ABB RobotStudio station: RobotStudio_PickAndGo.rspag

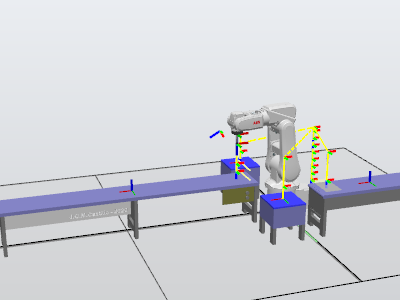
--- station ---
Station Project1 (saved by RobotStudio 24.4.11080.0)
Controller Controlador_1
  mechanical unit ROB_1: IRB120_3_58__01, 6 joints, base frame (0, 0, 0) mm
Layout (positions relative to the parent item):
  - IRB120_3_58__01 [mechanism, from %ABB.RobotStudio.Models.IRB120%\IRB120_3_58_G_01.rslib] at (0, 0, 0) mm; joint values [0.1232, 0.0796, -0.0396, 0, 1.5308, 0.1232] (rad or m)
  - CintaConveyor [protected smart component, left out]
  - CintaDescarga [protected smart component, left out]
  - Caja IZQ [protected smart component, left out]
  - Ventosa [protected smart component, left out]
  - Caja DER [protected smart component, left out]
Attachment: Ventosa is attached to IRB120_3_58__01 / Link6
Attachment: Workobject_Conveyor is attached to Belt
Attachment: Workobject_Mesa1 is attached to Tapa
Attachment: Workobject_CintaDescarga is attached to Cinta de transporte
Attachment: Workobject_Mesa2 is attached to Tapa
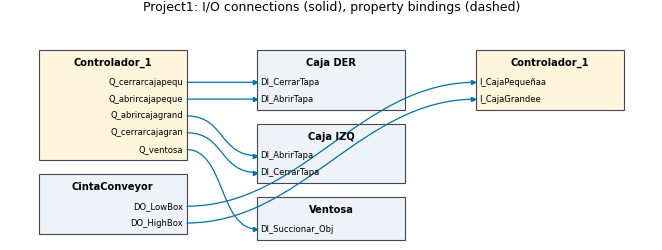
Station logic (signal -> signal, property => property):
  Controlador_1.Q_cerrarcajapequeña -> Caja DER.DI_CerrarTapa
  Controlador_1.Q_abrircajapequeña -> Caja DER.DI_AbrirTapa
  Controlador_1.Q_abrircajagrande -> Caja IZQ.DI_AbrirTapa
  Controlador_1.Q_cerrarcajagrande -> Caja IZQ.DI_CerrarTapa
  Controlador_1.Q_ventosa -> Ventosa.DI_Succionar_Objeto
  CintaConveyor.DO_LowBox -> Controlador_1.I_CajaPequeñaa
  CintaConveyor.DO_HighBox -> Controlador_1.I_CajaGrandee
Targets, tools, work objects and paths stored in the station and not in the controller backup, written as RAPID:
! task T_ROB1
MODULE Module1
  PROC setup()
    MoveJ Target_10,velocidad,z0,TCP_Ventosa\WObj:=wobj0;
  ENDPROC
ENDMODULE

! task T_ROB1
MODULE Rutinas_eventos
  PROC Paro_off()
    SetDO Q_Paro,0;
  ENDPROC
  PROC Paro_on()
    SetDO Q_Paro,1;
  ENDPROC
  PROC Power_Controladora()
    SetDO Q_Power_Controladora,1;
  ENDPROC
ENDMODULE


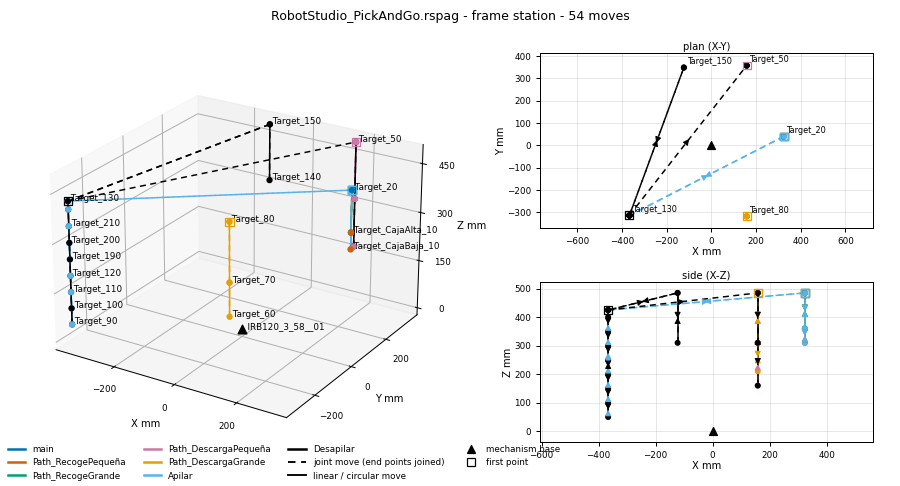
[picture p0: tool path of RobotStudio_PickAndGo.rspag in frame station, 54 of 54 moves have a stored position in this frame; points joined in program order, loops and branches not executed]
--- Controller Data/Controlador_1/RAPID/TASK1/PROGMOD/CalibData.mod ---
MODULE CalibData
    PERS tooldata TCP_Ventosa:=[TRUE,[[0,0,60],[1,0,0,0]],[0.1,[0,0,1],[1,0,0,0],0,0,0]];
    TASK PERS wobjdata Workobject_Conveyor:=[FALSE,TRUE,"",[[971.48,35.469,260],[1,0,0,0]],[[0,0,0],[1,0,0,0]]];
    TASK PERS wobjdata Workobject_Mesa1:=[FALSE,TRUE,"",[[158.333,357.694,230],[1,0,0,0]],[[0,0,0],[1,0,0,0]]];
    TASK PERS wobjdata Workobject_Mesa2:=[FALSE,TRUE,"",[[158.333,-317.306,230],[1,0,0,0]],[[0,0,0],[1,0,0,0]]];
    TASK PERS wobjdata Workobject_CintaDescarga:=[FALSE,TRUE,"",[[-411.761,348.55,260],[1,0,0,0]],[[0,0,0],[1,0,0,0]]];
    TASK PERS wobjdata Workobject_Apilar:=[FALSE,TRUE,"",[[-366.457,-313.205,0],[1,0,0,0]],[[0,0,0],[1,0,0,0]]];
ENDMODULE

--- Controller Data/Controlador_1/RAPID/TASK1/PROGMOD/Module1.mod ---
MODULE Module1
    VAR num contadorPiezas:=0;
    PERS num maximoPiezas:=2;
    PERS num tiempoEspera:=0;
    VAR speeddata velocidad := [1000,500,1000,500];
    PERS num vel;
    VAR bool marca_estado:=TRUE;
    VAR bool caja_o_cinta:=TRUE;
    VAR bool bloqueoDesapilar;
    VAR bool mensaje := TRUE;
    CONST robtarget Target_20:=[[-647.92,4.582,225],[-0.000000001,0,1,0],[0,0,0,0],[9E+09,9E+09,9E+09,9E+09,9E+09,9E+09]];
    CONST robtarget Target_CajaAlta_10:=[[-647.92,4.582,100],[-0.000000001,0,1,0],[0,0,0,0],[9E+09,9E+09,9E+09,9E+09,9E+09,9E+09]];
    CONST robtarget Target_CajaBaja_10:=[[-647.92,4.582,50],[-0.000000001,0,1,0],[0,0,0,0],[9E+09,9E+09,9E+09,9E+09,9E+09,9E+09]];
    CONST robtarget Target_50:=[[0.001,0,255],[-0.000000001,0,1,0],[0,0,0,0],[9E+09,9E+09,9E+09,9E+09,9E+09,9E+09]];
    CONST robtarget Target_40:=[[0.001,0,80],[-0.000000001,0,1,0],[0,0,0,0],[9E+09,9E+09,9E+09,9E+09,9E+09,9E+09]];
    CONST robtarget Target_30:=[[0.001,0,-70],[-0.000000001,0,1,0],[0,0,0,0],[9E+09,9E+09,9E+09,9E+09,9E+09,9E+09]];
    CONST robtarget Target_80:=[[0.001,0,255],[-0.000000001,0,1,0],[0,0,0,0],[9E+09,9E+09,9E+09,9E+09,9E+09,9E+09]];
    CONST robtarget Target_70:=[[0.001,0,80],[-0.000000001,0,1,0],[-1,-1,-1,0],[9E+09,9E+09,9E+09,9E+09,9E+09,9E+09]];
    CONST robtarget Target_60:=[[0.001,0,-20],[-0.000000001,0,1,0],[-1,-1,-1,0],[9E+09,9E+09,9E+09,9E+09,9E+09,9E+09]];
    CONST robtarget Target_130:=[[0,0,425],[-0.000000001,0,1,0],[-2,-1,-2,0],[9E+09,9E+09,9E+09,9E+09,9E+09,9E+09]];
    CONST robtarget Target_90:=[[0,0,50],[-0.000000001,0,1,0],[-2,-1,-2,0],[9E+09,9E+09,9E+09,9E+09,9E+09,9E+09]];
    CONST robtarget Target_100:=[[0,0,100],[-0.000000001,0,1,0],[-2,-1,-2,0],[9E+09,9E+09,9E+09,9E+09,9E+09,9E+09]];
    CONST robtarget Target_110:=[[0,0,150],[-0.000000001,0,1,0],[-2,-1,-2,0],[9E+09,9E+09,9E+09,9E+09,9E+09,9E+09]];
    CONST robtarget Target_120:=[[0,0,200],[-0.000000001,0,1,0],[-2,-1,-2,0],[9E+09,9E+09,9E+09,9E+09,9E+09,9E+09]];
    CONST robtarget Target_150:=[[288.994,0,225],[-0.000000001,0,1,0],[1,0,1,0],[9E+09,9E+09,9E+09,9E+09,9E+09,9E+09]];
    CONST robtarget Target_140:=[[288.994,0,50],[-0.000000001,0,1,0],[1,0,1,0],[9E+09,9E+09,9E+09,9E+09,9E+09,9E+09]];
    CONST robtarget Target_220:=[[0,0,400],[-0.000000001,0,1,0],[-2,-1,-2,0],[9E+09,9E+09,9E+09,9E+09,9E+09,9E+09]];
    CONST robtarget Target_190:=[[0,0,250],[-0.000000001,0,1,0],[-2,-1,-2,0],[9E+09,9E+09,9E+09,9E+09,9E+09,9E+09]];
    CONST robtarget Target_200:=[[0,0,300],[-0.000000001,0,1,0],[-2,-1,-2,0],[9E+09,9E+09,9E+09,9E+09,9E+09,9E+09]];
    CONST robtarget Target_210:=[[0,0,350],[-0.000000001,0,1,0],[-2,-1,-2,0],[9E+09,9E+09,9E+09,9E+09,9E+09,9E+09]];
    CONST robtarget Target_10:=[[416.3153533,0,564],[0.5,0,0.866025404,0],[0,0,0,0],[9E+09,9E+09,9E+09,9E+09,9E+09,9E+09]];

    PROC main()
        SetDO Q_Power_Controladora,0;
        IF mensaje = TRUE THEN
            TPWrite "Pulse Marcha para iniciar";
            TPWrite "Elija apilar o no apilar";
            WaitTime 5;
            TpShow tp_latest;
            TPErase;
            mensaje := FALSE;
        ENDIF
        MoveJ Target_20,velocidad,z0,TCP_Ventosa\WObj:=Workobject_Conveyor;
        WaitRob\InPos;
        WaitUntil marca_marcha = 1 OR Tecla = 1;
        velocidad := [vel,500,1000,500];
        IF I_CajaGrandee=0 AND I_CajaPequeñaa=1 AND interuptorEstado =0 procesoCajaPeq;
        IF I_CajaGrandee=0 AND I_CajaPequeñaa=1 AND interuptorEstado =1 AND bloqueoDesapilar=FALSE procesoApilar;
        IF I_CajaGrandee=0 AND I_CajaPequeñaa=1 AND interuptorEstado =1 AND bloqueoDesapilar=TRUE procesoDesapilar;
        IF I_CajaGrandee=1 AND I_CajaPequeñaa=1 procesoCajaGran;
    ENDPROC

    PROC procesoCajaPeq()
        Path_RecogePequeña;
        Path_DescargaPequeña;
    ENDPROC

    PROC procesoCajaGran()
        Path_RecogeGrande;
        Path_DescargaGrande;
    ENDPROC

    PROC procesoApilar()
        Apilar;
    ENDPROC

    PROC procesoDesapilar()
        Desapilar;
    ENDPROC

    PROC Path_RecogePequeña()
        MoveJ Target_20,velocidad,z0,TCP_Ventosa\WObj:=Workobject_Conveyor;
        MoveL Target_CajaAlta_10,velocidad,z0,TCP_Ventosa\WObj:=Workobject_Conveyor;
        MoveL Target_CajaBaja_10,velocidad,fine,TCP_Ventosa\WObj:=Workobject_Conveyor;
        SetDO Q_ventosa,1;
        WaitTime tiempoEspera;
        MoveJ Target_CajaAlta_10,velocidad,z0,TCP_Ventosa\WObj:=Workobject_Conveyor;
        MoveJ Target_20,velocidad,z0,TCP_Ventosa\WObj:=Workobject_Conveyor;
    ENDPROC

    PROC Path_RecogeGrande()
        MoveJ Target_20,velocidad,z0,TCP_Ventosa\WObj:=Workobject_Conveyor;
        MoveL Target_CajaAlta_10,velocidad,fine,TCP_Ventosa\WObj:=Workobject_Conveyor;
        SetDO Q_ventosa,1;
        WaitTime tiempoEspera;
        MoveJ Target_20,velocidad,z0,TCP_Ventosa\WObj:=Workobject_Conveyor;
    ENDPROC

    PROC Path_DescargaPequeña()
        MoveJ Target_50,velocidad,z0,TCP_Ventosa\WObj:=Workobject_Mesa1;
        MoveL Target_40,velocidad,fine,TCP_Ventosa\WObj:=Workobject_Mesa1;
        PulseDO Q_abrircajapequeña;
        MoveL Target_30,velocidad,fine,TCP_Ventosa\WObj:=Workobject_Mesa1;
        SetDO Q_ventosa,0;
        WaitTime tiempoEspera;
        MoveJ Target_40,velocidad,fine,TCP_Ventosa\WObj:=Workobject_Mesa1;
        PulseDO Q_cerrarcajapequeña;
        MoveJ Target_50,velocidad,z0,TCP_Ventosa\WObj:=Workobject_Mesa1;
    ENDPROC

    PROC Path_DescargaGrande()
        MoveJ Target_80,velocidad,z0,TCP_Ventosa\WObj:=Workobject_Mesa2;
        MoveL Target_70,velocidad,fine,TCP_Ventosa\WObj:=Workobject_Mesa2;
        PulseDO Q_abrircajagrande;
        MoveL Target_60,velocidad,fine,TCP_Ventosa\WObj:=Workobject_Mesa2;
        SetDO Q_ventosa,0;
        WaitTime tiempoEspera;
        MoveJ Target_70,velocidad,fine,TCP_Ventosa\WObj:=Workobject_Mesa2;
        PulseDO Q_cerrarcajagrande;
        MoveJ Target_80,velocidad,z0,TCP_Ventosa\WObj:=Workobject_Mesa2;
    ENDPROC

    PROC Apilar()
        MoveJ Target_20,velocidad,z0,TCP_Ventosa\WObj:=Workobject_Conveyor;
        MoveL Target_CajaAlta_10,velocidad,z0,TCP_Ventosa\WObj:=Workobject_Conveyor;
        MoveL Target_CajaBaja_10,velocidad,fine,TCP_Ventosa\WObj:=Workobject_Conveyor;
        SetDO Q_ventosa,1;
        WaitTime tiempoEspera;
        MoveL Target_CajaAlta_10,velocidad,z0,TCP_Ventosa\WObj:=Workobject_Conveyor;
        MoveJ Target_20,velocidad,z0,TCP_Ventosa\WObj:=Workobject_Conveyor;
        MoveJ Target_130,velocidad,z0,TCP_Ventosa\WObj:=Workobject_Apilar;
        IF contadorPiezas=0 THEN
            MoveL Target_90,velocidad,fine,TCP_Ventosa\WObj:=Workobject_Apilar;
        ELSEIF contadorPiezas=1 THEN
            MoveL Target_100,velocidad,fine,TCP_Ventosa\WObj:=Workobject_Apilar;
        ELSEIF contadorPiezas=2 THEN
            MoveL Target_110,velocidad,fine,TCP_Ventosa\WObj:=Workobject_Apilar;
        ELSEIF contadorPiezas=3 THEN
            MoveL Target_120,velocidad,fine,TCP_Ventosa\WObj:=Workobject_Apilar;
        ELSEIF contadorPiezas=4 THEN
            MoveL Target_190,velocidad,fine,TCP_Ventosa\WObj:=Workobject_Apilar;
        ELSEIF contadorPiezas=5 THEN
            MoveL Target_200,velocidad,fine,TCP_Ventosa\WObj:=Workobject_Apilar;
        ELSEIF contadorPiezas=6 THEN
            MoveL Target_210,velocidad,fine,TCP_Ventosa\WObj:=Workobject_Apilar;
        ELSEIF contadorPiezas=7 THEN
            MoveL Target_220,velocidad,fine,TCP_Ventosa\WObj:=Workobject_Apilar;
        ENDIF
        SetDO Q_ventosa,0;
        WaitTime tiempoEspera;
        MoveJ Target_130,velocidad,z0,TCP_Ventosa\WObj:=Workobject_Apilar;

        IF contadorPiezas<8 THEN
            contadorPiezas:=contadorPiezas+1;
        ENDIF

        IF contadorPiezas=maximoPiezas THEN
            MoveJ Target_130,velocidad,z0,TCP_Ventosa\WObj:=Workobject_Apilar;
            MoveJ Target_20,velocidad,fine,TCP_Ventosa\WObj:=Workobject_Conveyor;
            SetDO Alerta,1;
            WaitUntil PulsadorReanudar=1;
            IF PulsadorReanudar =1 THEN
                IF CajaOCinta=1 THEN
                    caja_o_cinta:=TRUE;
                ENDIF
                IF CajaOCinta =0 THEN
                    caja_o_cinta:=FALSE;
                ENDIF
                bloqueoDesapilar:=TRUE;
                SetDO Alerta,0;
            ENDIF
        ENDIF
    ENDPROC

    PROC Desapilar()
        MoveJ Target_130,velocidad,fine,TCP_Ventosa\WObj:=Workobject_Apilar;
        IF contadorPiezas=8 THEN
            MoveL Target_220,velocidad,fine,TCP_Ventosa\WObj:=Workobject_Apilar;
            SetDO Q_ventosa,1;
            WaitTime tiempoEspera;
        ELSEIF contadorPiezas=7 THEN
            MoveL Target_210,velocidad,fine,TCP_Ventosa\WObj:=Workobject_Apilar;
            SetDO Q_ventosa,1;
            WaitTime tiempoEspera;
        ELSEIF contadorPiezas=6 THEN
            MoveL Target_200,velocidad,fine,TCP_Ventosa\WObj:=Workobject_Apilar;
            SetDO Q_ventosa,1;
            WaitTime tiempoEspera;
        ELSEIF contadorPiezas=5 THEN
            MoveL Target_190,velocidad,fine,TCP_Ventosa\WObj:=Workobject_Apilar;
            SetDO Q_ventosa,1;
            WaitTime tiempoEspera;
        ELSEIF contadorPiezas=4 THEN
            MoveL Target_120,velocidad,fine,TCP_Ventosa\WObj:=Workobject_Apilar;
            SetDO Q_ventosa,1;
            WaitTime tiempoEspera;
        ELSEIF contadorPiezas=3 THEN
            MoveL Target_110,velocidad,fine,TCP_Ventosa\WObj:=Workobject_Apilar;
            SetDO Q_ventosa,1;
            WaitTime tiempoEspera;
        ELSEIF contadorPiezas=2 THEN
            MoveL Target_100,velocidad,fine,TCP_Ventosa\WObj:=Workobject_Apilar;
            SetDO Q_ventosa,1;
            WaitTime tiempoEspera;
        ELSEIF contadorPiezas=1 THEN
            MoveL Target_90,velocidad,fine,TCP_Ventosa\WObj:=Workobject_Apilar;
            SetDO Q_ventosa,1;
            WaitTime tiempoEspera;
        ENDIF

        IF caja_o_cinta=TRUE THEN
            MoveJ Target_130,velocidad,z0,TCP_Ventosa\WObj:=Workobject_Apilar;
            MoveJ Target_150,velocidad,z0,TCP_Ventosa\WObj:=Workobject_CintaDescarga;
            MoveL Target_140,velocidad,fine,TCP_Ventosa\WObj:=Workobject_CintaDescarga;
            SetDO Q_ventosa,0;
            WaitTime tiempoEspera;
            MoveJ Target_150,velocidad,z0,TCP_Ventosa\WObj:=Workobject_CintaDescarga;
        ENDIF

        IF caja_o_cinta=FALSE THEN
            MoveJ Target_130,velocidad,z0,TCP_Ventosa\WObj:=Workobject_Apilar;
            MoveJ Target_50,velocidad,z0,TCP_Ventosa\WObj:=Workobject_Mesa1;
            MoveL Target_40,velocidad,fine,TCP_Ventosa\WObj:=Workobject_Mesa1;
            PulseDO Q_abrircajapequeña;
            MoveL Target_30,velocidad,fine,TCP_Ventosa\WObj:=Workobject_Mesa1;
            SetDO Q_ventosa,0;
            WaitTime tiempoEspera;
            MoveJ Target_50,velocidad,z0,TCP_Ventosa\WObj:=Workobject_Mesa1;
            WaitRob\InPos;
            PulseDO Q_cerrarcajapequeña;
        ENDIF

        IF contadorPiezas>0 THEN
            contadorPiezas:=contadorPiezas-1;
        ENDIF

        IF contadorPiezas=0 THEN
            bloqueoDesapilar:=FALSE;
        ENDIF

    ENDPROC
ENDMODULE

--- Controller Data/Controlador_1/RAPID/TASK1/PROGMOD/RsTempModule.mod ---
MODULE RsTempModule
ENDMODULE

--- Controller Data/Controlador_1/RAPID/TASK1/PROGMOD/Rutinas_eventos.mod ---
MODULE Rutinas_eventos
    PROC Marcha()
        SetDO Q_Power_Controladora,1;
    ENDPROC
ENDMODULE

--- Controller Data/Controlador_1/SYSPAR/EIO.cfg ---
EIO:CFG_1.0:6:1::
#
INDUSTRIAL_NETWORK:

      -Name "DeviceNet" -Label "DeviceNet Master/Slave Network" -Address "2"
#
DEVICENET_DEVICE:

      -Name "d652" -VendorName "ABB Robotics" -ProductName "24 VDC I/O Device"\
      -Label "DSQC 652 24 VDC I/O Device" -Address 10 -ProductCode 26\
      -DeviceType 7 -ConnectionType "COS" -OutputSize 2 -InputSize 2
#
DEVICENET_INTERNAL_DEVICE:

      -Name "DN_Internal_Device" -VendorName "ABB Robotics"\
      -ProductName "DeviceNet Internal Slave Device"
#
EIO_SIGNAL:

      -Name "I_cajagrande" -SignalType "DI"

      -Name "I_cajapequeña" -SignalType "DI"

      -Name "Q_ventosa" -SignalType "DO"

      -Name "Q_abrircajagrande" -SignalType "DO"

      -Name "Q_cerrarcajagrande" -SignalType "DO"

      -Name "Q_abrircajapequeña" -SignalType "DO"

      -Name "Q_cerrarcajapequeña" -SignalType "DO"

      -Name "I_CajaGrandee" -SignalType "DI"

      -Name "I_CajaPequeñaa" -SignalType "DI"

      -Name "PulsadorReanudar" -SignalType "DO" -Access "All"

      -Name "CajaOCinta" -SignalType "DO" -Access "All"

      -Name "InteruptorEstado" -SignalType "DO" -Access "All"

      -Name "Alerta" -SignalType "DO" -Device "d652" -DeviceMap "4"\
      -Access "All"

      -Name "marca_marcha" -SignalType "DO" -Access "All"

      -Name "Q_Power_Controladora" -SignalType "DO"

      -Name "Tecla" -SignalType "DO" -Device "d652" -DeviceMap "7" -Access "All"
